FUNCTION_BLOCK E_MERGE4 (* Basic Function Block Type *)
  (* Standard: 61499-2 *)
  (* Version 0.0, 11/14/2025, vv263, Template *)
  PACKAGE Main;
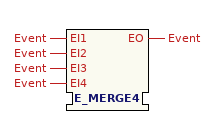
  EVENT_INPUT
    EI1; (* Initialization Request *)
    EI2; (* Normal Execution Request *)
    EI3;
    EI4;
  END_EVENT
  EVENT_OUTPUT
    EO; (* Initialization Confirm *)
  END_EVENT
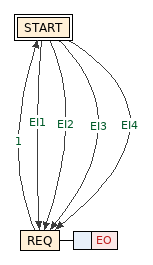
  EC_STATES
    START; (* Initial State *)
    REQ : -> EO; (* Normal execution *)
  END_STATES
  EC_TRANSITIONS
    START TO REQ := EI1;
    REQ TO START := 1;
    START TO REQ := EI2;
    START TO REQ := EI3;
    START TO REQ := EI4;
  END_TRANSITIONS
  ALGORITHM INIT IN ST: (* Initialization algorithm *)
;
  END_ALGORITHM
  ALGORITHM REQ IN ST: (* Normally executed algorithm *)
;
  END_ALGORITHM
END_FUNCTION_BLOCK
